Staubli VAL3: JointTrajPtFull.dtx

public Body body
  [0]
    num accelerations[10]
      [0] = 100
      [1] = 100
    num positions[10]
      [0] = 0.178024
      [1] = 0.405265
      [2] = 0.788191
      [3] = 0.125664
      [4] = 0.444186
      [5] = -0.149575
    num robotId = 92
    num sequence
    num time = 23.78133
    num validFields = 14
    num velocities[10] = 100
public Header header
  [0]
    num nMsgType = 14
    num nCommType = 3
    num nReplyCode = 1
public Prefix prefix
  [0]
    num nLength = 148
mdesc mNomSpeed
